TEXTLIST TextList_Moteurs
  0 = '' | FR: 'Reset Moteur' | EN: 'Motor Reset'
  1 = '' | FR: 'Reset Position' | EN: 'Position Reset'
  2 = '' | FR: 'Dévalidation' | EN: 'Devalidation'
  3 = '' | FR: 'Compteur de\nbalayages' | EN: 'Sweepings\nCounter'
  4 = '' | FR: 'Aller en position de transfert' | EN: 'Go to transfer position'
  5 = '' | FR: 'Position\nBasse' | EN: 'Low\nPosition'
  6 = '' | FR: 'Position\nHaute' | EN: 'High\nPosition'
  7 = '' | FR: 'Vitesse' | EN: 'Speed'
  8 = '' | FR: 'Poste' | EN: 'Station'
  9 = '' | FR: 'Distance' | EN: 'Distance'
  10 = '' | FR: 'De' | EN: 'From'
  11 = '' | FR: 'Réf.' | EN: 'Homed'
  12 = '' | FR: 'Position' | EN: 'Position'
  13 = '' | FR: 'Poste sélectionné' | EN: 'Selected station'
  14 = '' | FR: 'Référence sélectionnée' | EN: 'Selected reference'
  15 = '' | FR: 'Consignes' | EN: 'Setpoints'
  16 = '' | FR: 'Amplitude balayage' | EN: 'Sweeping amplitude'
  17 = '' | FR: 'Accélération' | EN: 'Acceleration'
  18 = '' | FR: 'Décélération' | EN: 'Deceleration'
  19 = '' | FR: 'Avec prise\nde référence' | EN: 'With\nHoming'
  20 = '' | FR: 'Sans prise\nde référence' | EN: 'Without\nHoming'
  21 = '' | FR: 'Départ centré' | EN: 'Centered start'
  22 = '' | FR: 'Départ déporté' | EN: 'Deported start'
   = ''
END_TEXTLIST

(* stored: Version 1.1.0.1, ProductVersion 3.1.4024.10
   TextList TextList_Moteurs: Id {2f8b6983-5840-4848-bb0c-71f7dfad1cb1} *)
